// TIA Portal V17 export
// export: Created 2021-12-03T08:13:08.6951796Z, ExportSetting WithDefaults, DisplayName Totally Integrated Automation Portal, DisplayVersion V17, DisplayName TIA Portal Openness, DisplayVersion V17, DisplayName TIA Portal Version Control Interface, DisplayVersion V17, DisplayName STEP 7 Professional, DisplayVersion V17, DisplayName STEP 7 Safety, DisplayVersion V17, DisplayName WinCC Advanced, DisplayVersion V17
DATA_BLOCK "GDB_Faults"   // DB40
VERSION : 0.1
// stored: AutoNumber false, IsOnlyStoredInLoadMemory false, IsWriteProtectedInAS false
   VAR
      CirBrk24VFb { ExternalVisible := 'False'} : Struct
         I_BrPow1Flt { ExternalVisible := 'False'} : Bool := false;   // Breaker Powersupply 1 24VDC Fault
         I_BrPow2Flt { ExternalVisible := 'False'} : Bool := false;   // Breaker Powersupply 2 24VDC Fault
         I_SitopPow1Flt { ExternalVisible := 'False'} : Bool;   // Sitop Diagnose Modul Powersupply 1 Failure
         I_SitopPow2Flt { ExternalVisible := 'False'} : Bool;   // Sitop Diagnose Modul Powersupply 2 Failure
      END_STRUCT;
      CirBrk220VFb { ExternalVisible := 'False'} : Struct
         I_BrLigSrvFlt { ExternalVisible := 'False'} : Bool;   // Breaker Light and Service Outlet Fault
         I_BrAccConFlt { ExternalVisible := 'False'} : Bool;   // Breaker Accelerator Console Fault
         I_BrXRayUnitFlt { ExternalVisible := 'False'} : Bool;   // Breaker X-Ray Unit Fault
         I_BrPowPlcFlt { ExternalVisible := 'False'} : Bool;   // Breaker Powersupply PS307 (PLC) Fault
         I_BrMod1PFlt { ExternalVisible := 'False'} : Bool;   // Breaker Modulator 230 VAC Fault
      END_STRUCT;
      CirBrk380VFb { ExternalVisible := 'False'} : Struct
         I_BrModFlt { ExternalVisible := 'False'} : Bool;   // Breaker Modulator Fault
         I_BrChilFlt { ExternalVisible := 'False'} : Bool;   // Breaker Chiller Fault
         I_BrFrqConvFlt { ExternalVisible := 'False'} : Bool;   // Breaker Frequnce Converter Conveyor Fault
      END_STRUCT;
      FeedBackControl { ExternalVisible := 'False'} : Struct
         ModCont400_Err { ExternalVisible := 'False'} : Bool;   // Ошибка включения модулятора 400v
         ModCont230_Err { ExternalVisible := 'False'} : Bool;   // Ошибка включения модулятора 230v
         ChillCont_Err { ExternalVisible := 'False'} : Bool;   // Ошибка включения чиллера
         AccCont_Err { ExternalVisible := 'False'} : Bool;   // Ошибка включения ускорителя
         ConvCont_Err { ExternalVisible := 'False'} : Bool;   // Ошибка включения конвеера
      END_STRUCT;
      EmStBt { ExternalVisible := 'False'} : Struct
         P1EmStp_Sv { ExternalVisible := 'False'} : Bool;   // Аварийная кнопка Пульт Р1
         P2EmStp_Sv { ExternalVisible := 'False'} : Bool;   // Аварийная кнопка Пульт Р2
         P3EmStp_Sv { ExternalVisible := 'False'} : Bool;   // Аварийная кнопка Пульт Р3
         AccEmStp_Sv { ExternalVisible := 'False'} : Bool;   // Аварийная кнопка ускорителя
         DosimEmStp_Sv { ExternalVisible := 'False'} : Bool;   // Дозиметр
         PerOpnIllegal { ExternalVisible := 'False'} : Bool;   // Периметр разорван не легально
      END_STRUCT;
      Conveyer { ExternalVisible := 'False'} : Struct
         FrqConv { ExternalVisible := 'False'} : Bool;   // Ошибка частотного преобразователя
         FrqConv_Ack { ExternalVisible := 'False'} : Bool;
         CycleTime { ExternalVisible := 'False'} : Bool;   // Превышено время сканирования
         CycleTime_Ack { ExternalVisible := 'False'} : Bool;
         IntrptCycl { ExternalVisible := 'False'} : Bool;   // Цикл прерван
         IntrptCycl_Ack { ExternalVisible := 'False'} : Bool;
         Sns { ExternalVisible := 'False'} : Bool;   // Одновременное срабатывание датчиков
      END_STRUCT;
      DetLine { ExternalVisible := 'False'} : Struct
         NotCon { ExternalVisible := 'False'} : Bool;   // Нет соединения с детекторной линейкой
      END_STRUCT;
      Com_Err { ExternalVisible := 'False'} : Bool;   // Общая ошибка
   END_VAR
BEGIN
END_DATA_BLOCK
